FUNCTION_BLOCK Led
VAR
	_state	AT%M* : BOOL;
END_VAR

PROPERTY State : BOOL
GET
State := _state;
END_GET
SET
_state := State;
END_SET
END_PROPERTY

END_FUNCTION_BLOCK

(* stored: Version 1.1.0.1, ProductVersion 3.1.4024.12
   POU Led: Id {5192deaf-a571-4c56-a193-61331a8e0b7c}, SpecialFunc None
   Property State: Id {d42ba43d-b562-46aa-bef9-a5c2dcfb7fcb}
   Get Get: Id {ce5c1849-9ed5-42f0-923d-bafeb1f9a12a}
   Set Set: Id {e2261ee8-000f-442a-9440-c1ecbed6ff40} *)
